(* CODESYS project transformMatrix.project

Project tree, tasks and I/O mapping:
  Device : CODESYS Control Win V3 x64, 3S - Smart Software Solutions GmbH, version 3.5.12.0
    application Application
      libraries: Standard, * (System); SM3_Math, 4.3.0.0 (3S - Smart Software Solutions GmbH)
      task MainTask (cyclic, interval t#20ms, priority 1) calls PLC_PRG
      program PLC_PRG [ST]
      data type DUT_userFrame
      data type DUT_position
      function block UserToBase [ST]
*)

// Device/Application/DUT_userFrame
TYPE DUT_userFrame :
STRUCT
	X : DINT;//单位0.01mm
	Y : DINT;
	Z : DINT;
	A : DINT;
	B : DINT;
	C : DINT; //绕Z轴的转动角度 单位0.01度
END_STRUCT
END_TYPE

// Device/Application/DUT_position
TYPE DUT_position :
STRUCT
	X : DINT;//单位0.01mm
	Y : DINT;
	Z : DINT;
	A : DINT;
	B : DINT;
	C : DINT;//绕Z轴的转动角度 单位0.01度
END_STRUCT
END_TYPE

// Device/Application/PLC_PRG
PROGRAM PLC_PRG
VAR
	pos : DUT_position;
	userFrame : DUT_userFrame;
	answer : DUT_position;
	UB : UserToBase;
END_VAR

pos.X:=100;
pos.Y:=100;
pos.z:=3;

userFrame.X:=0;
userFrame.Y:=0;
userFrame.Z:=1;

userFrame.C:=-4500;


UB(pos:= pos, userFrame:= userFrame, basePos=>answer );

END_PROGRAM

// Device/Application/UserToBase
FUNCTION_BLOCK UserToBase
VAR_INPUT
	pos : DUT_position;//待计算输入点，在用户坐标下的值 
	userFrame : DUT_userFrame;//输入的用户坐标
END_VAR
VAR_OUTPUT
	basePos : DUT_position;//计算结果值
END_VAR
VAR
	temp_UF_C : LREAL;//用户坐标系绕Z轴转动的角度C
	transMatrix : ARRAY[1..4,1..4] OF LREAL;//变换矩阵
	temp_Vector : ARRAY[1..4] OF DINT;
	
	temp_sum : ARRAY[1..4] OF LREAL;
	
	i,j:int;//循环标志向量 i为行，j为列
END_VAR

VAR CONSTANT
	Deg2Rad : LREAL := smc_pi/180;
	Rad2Deg : LREAL := 180/smc_pi;
END_VAR

basePos.A := 0;//A,B在Gantry机器人中用不上
basePos.B :=0;
basePos.C := userFrame.C + pos.C;

temp_UF_C :=  userFrame.C/100 * Deg2Rad;//转成度再转成弧度

(*
	平面坐标系变换矩阵 乘       用户坐标下的代求点向量
	|cos(θ)  -sin(θ)  0  X0|     | Xu|   
	|sin(θ)   cos(θ)  0  Y0|   * | Zu| 
	|0         0      1  Z0|     | Yu|
    |0         0      0  1 |     | 1 |
*)
//绕Z轴转换矩阵赋值
transMatrix[1,1] := COS(temp_UF_C);   
transMatrix[1,2] := -SIN(temp_UF_C);
transMatrix[1,3] := 0;
transMatrix[1,4] := userFrame.X;

transMatrix[2,1] := SIN(temp_UF_C);
transMatrix[2,2] := COS(temp_UF_C);
transMatrix[2,3] := 0;
transMatrix[2,4] := userFrame.Y;

transMatrix[3,1] := 0;
transMatrix[3,2] := 0;
transMatrix[3,3] := 1;
transMatrix[3,4] := userFrame.Z;

transMatrix[4,1] := 0;
transMatrix[4,2] := 0;
transMatrix[4,3] := 0;
transMatrix[4,4] := 1;


//用户坐标下的待求点向量复制
temp_Vector[1]:=pos.X;
temp_Vector[2]:=pos.Y;
temp_Vector[3]:=pos.Z;
temp_Vector[4]:=1;

FOR i :=1 TO 4 DO
	temp_sum[i]:=0;
	FOR j:=1 TO 4 DO
		temp_sum[i]:=temp_sum[i]+transMatrix[i,j]*temp_Vector[j];
	END_FOR
END_FOR

basePos.X := LREAL_TO_DINT(temp_sum[1]);
basePos.Y := LREAL_TO_DINT(temp_sum[2]);
basePos.Z := LREAL_TO_DINT(temp_sum[3]);

END_FUNCTION_BLOCK
